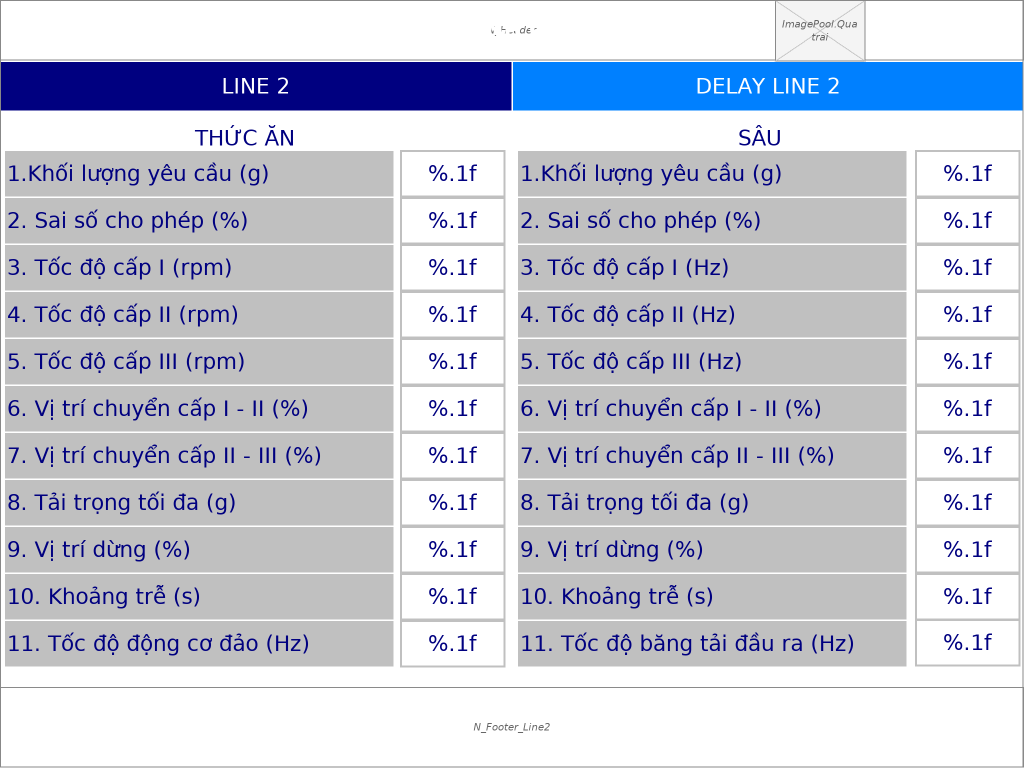
VISUALIZATION N_Setting_Line2  // 1024x768
    Frame (0,687 1024x80)
        shows N_Footer_Line2()
    Frame (0,0 1024x60)
        shows N_Header()
    Textfield (353,5 400x50), "MÀN HÌNH CÀI ĐẶT LINE 2"
    Textfield (170,120 150x36), "THỨC ĂN"
    Textfield (720,120 80x36), "SÂU"
    Rectangle (0,61 512x50), "LINE 2"
        OnMouseClick: change screen: N_Setting_Line2
    Rectangle (512,61 512x50), "DELAY LINE 2"
        OnMouseClick: change screen: N_Setting_Delay_JarSupply2
    Rectangle (517,150 390x47), "1.Khối lượng yêu cầu (g)"
    Rectangle (517,197 390x47), "2. Sai số cho phép (%)"
    Rectangle (517,244 390x47), "3. Tốc độ cấp I (Hz)"
    Rectangle (517,291 390x47), "4. Tốc độ cấp II (Hz)"
    Rectangle (517,385 390x47), "6. Vị trí chuyển cấp I - II (%)"
    Rectangle (517,479 390x47), "8. Tải trọng tối đa (g)"
    Rectangle (517,338 390x47), "5. Tốc độ cấp III (Hz)"
    Rectangle (517,432 390x47), "7. Vị trí chuyển cấp II - III (%)"
    Rectangle (517,573 390x47), "10. Khoảng trễ (s)"
    Rectangle (517,526 390x47), "9. Vị trí dừng (%)"
    Textfield (915,150 105x47), "%.1f", text variable: PR_Line02.fDerisedWeight_Worm
        OnMouseClick: write PR_Line02.fDerisedWeight_Worm via VisuDialogs.Numpad
    Textfield (915,197 105x47), "%.1f", text variable: PR_Line02.fDelta_Worm
        OnMouseClick: write PR_Line02.fDelta_Worm via VisuDialogs.Numpad
    Textfield (915,244 105x47), "%.1f", text variable: PR_Line02.fFast_Speed_vibrating_funnel
        OnMouseClick: write PR_Line02.fFast_Speed_vibrating_funnel via VisuDialogs.Numpad
    Textfield (915,291 105x47), "%.1f", text variable: PR_Line02.fSlow_Speed_vibrating_funnel_1
        OnMouseClick: write PR_Line02.fSlow_Speed_vibrating_funnel_1 via VisuDialogs.Numpad
    Textfield (915,338 105x47), "%.1f", text variable: PR_Line02.fSlow_Speed_vibrating_funnel_2
        OnMouseClick: write PR_Line02.fSlow_Speed_vibrating_funnel_2 via VisuDialogs.Numpad
    Textfield (915,385 105x47), "%.1f", text variable: PR_Line02.fChangeMode_Worm_1
        OnMouseClick: write PR_Line02.fChangeMode_Worm_1 via VisuDialogs.Numpad
    Textfield (915,432 105x47), "%.1f", text variable: PR_Line02.fChangeMode_Worm_2
        OnMouseClick: write PR_Line02.fChangeMode_Worm_2 via VisuDialogs.Numpad
    Textfield (915,479 105x47), "%.1f", text variable: PR_Line02.fMaxWeight_Worm
        OnMouseClick: write PR_Line02.fMaxWeight_Worm via VisuDialogs.Numpad
    Textfield (915,526 105x47), "%.1f", text variable: PR_Line02.fPerStop_Worm
        OnMouseClick: write PR_Line02.fPerStop_Worm via VisuDialogs.Numpad
    Textfield (915,573 105x47), "%.1f", text variable: PR_Line02.fTimer_Check_Worm
        OnMouseClick: write PR_Line02.fTimer_Check_Worm via VisuDialogs.Numpad
    Rectangle (4,150 390x47), "1.Khối lượng yêu cầu (g)"
    Rectangle (4,197 390x47), "2. Sai số cho phép (%)"
    Rectangle (4,244 390x47), "3. Tốc độ cấp I (rpm)"
    Rectangle (4,291 390x47), "4. Tốc độ cấp II (rpm)"
    Rectangle (4,385 390x47), "6. Vị trí chuyển cấp I - II (%)"
    Rectangle (4,479 390x47), "8. Tải trọng tối đa (g)"
    Rectangle (4,338 390x47), "5. Tốc độ cấp III (rpm)"
    Rectangle (4,432 390x47), "7. Vị trí chuyển cấp II - III (%)"
    Rectangle (4,573 390x47), "10. Khoảng trễ (s)"
    Rectangle (4,526 390x47), "9. Vị trí dừng (%)"
    Rectangle (4,620 390x47), "11. Tốc độ động cơ đảo (Hz)"
    Textfield (400,150 105x47), "%.1f", text variable: PR_Line02.fDerisedWeight_Food
        OnMouseClick: write PR_Line02.fDerisedWeight_Food via VisuDialogs.Numpad
    Textfield (400,197 105x47), "%.1f", text variable: PR_Line02.fDelta_Food
        OnMouseClick: write PR_Line02.fDelta_Food via VisuDialogs.Numpad
    Textfield (400,244 105x47), "%.1f", text variable: PR_Line02.fFast_Speed
        OnMouseClick: write PR_Line02.fFast_Speed via VisuDialogs.Numpad
    Textfield (400,291 105x47), "%.1f", text variable: PR_Line02.fSlow_Speed_1
        OnMouseClick: write PR_Line02.fSlow_Speed_1 via VisuDialogs.Numpad
    Textfield (400,338 105x47), "%.1f", text variable: PR_Line02.fSlow_Speed_2
        OnMouseClick: write PR_Line02.fSlow_Speed_2 via VisuDialogs.Numpad
    Textfield (400,385 105x47), "%.1f", text variable: PR_Line02.fChangeMode_Food_1
        OnMouseClick: write PR_Line02.fChangeMode_Food_1 via VisuDialogs.Numpad
    Textfield (400,432 105x47), "%.1f", text variable: PR_Line02.fChangeMode_Food_2
        OnMouseClick: write PR_Line02.fChangeMode_Food_2 via VisuDialogs.Numpad
    Textfield (400,479 105x47), "%.1f", text variable: PR_Line02.fMaxWeight_Food
        OnMouseClick: write PR_Line02.fMaxWeight_Food via VisuDialogs.Numpad
    Textfield (400,526 105x47), "%.1f", text variable: PR_Line02.fPerStop_Food
        OnMouseClick: write PR_Line02.fPerStop_Food via VisuDialogs.Numpad
    Textfield (400,573 105x47), "%.1f", text variable: PR_Line02.fTimer_Check_Food
        OnMouseClick: write PR_Line02.fTimer_Check_Food via VisuDialogs.Numpad
    Textfield (400,620 105x47), "%.1f", text variable: PR_Line02.fSpeed_motor_mixer
        OnMouseClick: write PR_Line02.fSpeed_motor_mixer via VisuDialogs.Numpad
    Image (775,0 90x61), image: ImagePool.Qua trai
        OnMouseClick: change screen: N_Setting_Line1
    Rectangle (517,620 390x47), "11. Tốc độ băng tải đầu ra (Hz)"
    Textfield (915,619 105x47), "%.1f", text variable: PR_Conveyor_Out.fSpeed_Conveyor
        OnMouseClick: write PR_Conveyor_Out.fSpeed_Conveyor via VisuDialogs.Numpad
END_VISUALIZATION

(* stored: Version 1.1.0.1, ProductVersion 3.1.4024.12
   Visu N_Setting_Line2: Id {49afb4c4-5ed4-4a14-8365-0efa4c37343e} *)
